FUNCTION F_ParseRawVarint32 : HRESULT
VAR_IN_OUT CONSTANT
    aBuffer : ARRAY [*] OF BYTE;
END_VAR
VAR_IN_OUT
    stState : ST_ParserInternalState;
END_VAR
VAR_INPUT
    anyVarInt32Result : ANY_INT;
END_VAR
VAR 
    bTmpByte        : BYTE;
    nResult         : UDINT;
    nShift          : UINT := 1;
    i               : UINT;
END_VAR

IF anyVarInt32Result.diSize > SIZEOF(UDINT) THEN
    F_ParseRawVarint32 := stState.eParserErrorCode := E_ParserErrorCode.InvalidDataType;     
    RETURN; 
END_IF

IF UPPER_BOUND(aBuffer,1) > TO_DINT(stState.nBufferSize) THEN
    F_ParseRawVarint32 := stState.eParserErrorCode := E_ParserErrorCode.TruncatedMessage;     
    RETURN; 
END_IF

bTmpByte := aBuffer[stState.nBufferPos];

stState.nBufferPos := stState.nBufferPos + 1;

IF bTmpByte < 16#80 THEN
    nResult := TO_UDINT(bTmpByte);
    MEMMOVE(destAddr:= anyVarInt32Result.pValue, srcAddr:= ADR(nResult), SIZEOF(nResult));
    RETURN;
END_IF 

nResult := bTmpByte AND 16#7F;

{warning 'TODO: MalformedVarInt needs to be compared with C# protobuf}

WHILE (bTmpByte > 16#7F AND TO_DINT(stState.nBufferPos) <= UPPER_BOUND(aBuffer, 1) AND nShift < 5) DO
    bTmpByte := aBuffer[stState.nBufferPos];
    
    // MalformedVarInt when we encounter zero value, but MSB was set last iteration.
    IF bTmpByte = 0 THEN
        stState.eParserErrorCode := E_ParserErrorCode.MalformedVarInt;
        JMP _ERROR_FUNCTION;
    END_IF
    
    IF nShift = 4 AND bTmpByte >= 16#80 THEN        
        // Likely a negative encoded value, should have been encoded as SInt32 instead (protofile)...
        nResult := nResult OR SHL((bTmpByte AND 16#7F), nShift * 7);
        FOR i:= 0 TO 5 DO
            // Discard upper 32 bits.
            F_ParseRawVarint32 := F_ReadRawByte(aBuffer, stState, nByte=> bTmpByte);
            IF bTmpByte < 16#80 THEN                
                JMP _END_FUNCTION;
            END_IF
        END_FOR
        stState.eParserErrorCode := E_ParserErrorCode.MalformedVarInt;
        JMP _ERROR_FUNCTION;
    
    END_IF
        
    nResult := nResult OR SHL((bTmpByte AND 16#7F), nShift * 7); 
    nShift := nShift + 1; 
    stState.nBufferPos := stState.nBufferPos + 1;
END_WHILE 

_END_FUNCTION:
MEMMOVE(destAddr:= anyVarInt32Result.pValue, srcAddr:= ADR(nResult), SIZEOF(nResult));
F_ParseRawVarint32 := S_OK;
RETURN;

_ERROR_FUNCTION:
F_ParseRawVarint32 := stState.eParserErrorCode;
stState.bError := TRUE;
nResult := 0;
RETURN;

END_FUNCTION

(* stored: Version 1.1.0.1
   POU F_ParseRawVarint32: Id {51c6c8a1-a14a-4443-b331-fa1787d7bb62}, SpecialFunc None *)
